(* PLC project Unnamed, Unknown Unnamed 1 *)
(* stored: creationDateTime 2022-12-13T19:44:02, modificationDateTime 2022-12-13T20:10:28 *)

PROGRAM water_tank
  VAR_INPUT
    High : BOOL;
    Low : BOOL;
  END_VAR
  VAR_OUTPUT
    Valve_In : BOOL;
    Valve_Out : BOOL;
  END_VAR
  VAR_INPUT
    Start : BOOL;
    Stop : BOOL;
  END_VAR
  VAR
    Master : BOOL;
  END_VAR

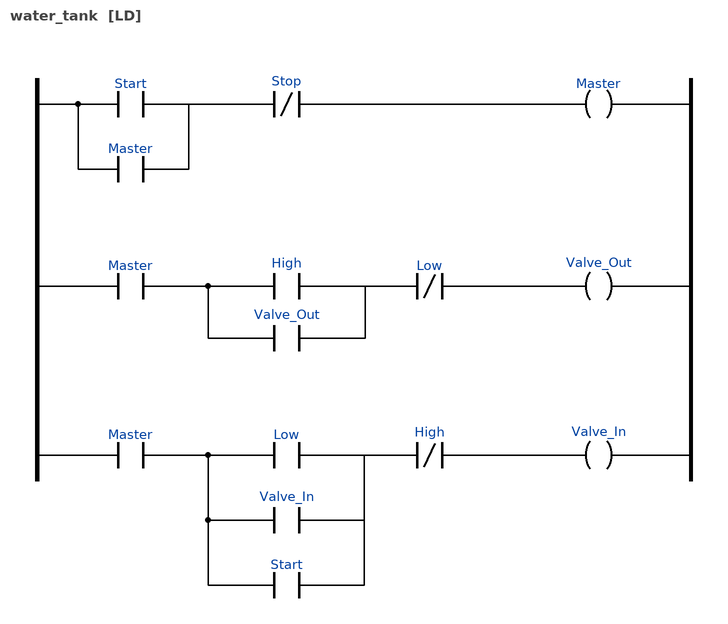
(* LD diagram, written out as Structured Text *)
Master := (Start OR Master) AND NOT Stop;
Valve_Out := Master AND (High OR Valve_Out) AND NOT Low;
Valve_In := Master AND (Low OR Valve_In OR Start) AND NOT High;
END_PROGRAM

CONFIGURATION Config0
  RESOURCE Res0 ON PLC
    TASK task0(INTERVAL := T#20ms, PRIORITY := 0);
    PROGRAM instance0 WITH task0 : water_tank;
  END_RESOURCE
END_CONFIGURATION
